Staubli VAL3: MotionMode.dtx

public num JOINT_TRAJ
public num VELOCITY_CTRL
public num INVALID
